(* IEC 61131-3 sources: CodesysTest/alpha/export/FBs/Components/BagOpenFingers/FB_BagOpenFingers.pou, 1 file *)

(* ---- FB_BagOpenFingers.pou.st ---- *)
(*#-#-#-#-#-#-#-#-#-#---Declaration---#-#-#-#-#-#-#-#-#-#-#-#-#*)

FUNCTION_BLOCK FB_BagOpenFingers EXTENDS FB_BaseComponent
VAR_INPUT
END_VAR
VAR_OUTPUT
    releaseOutput : BOOL;
	grabOutput : BOOL;
END_VAR
VAR
    _releaseCommand : BOOL;
    _grabCommand : BOOL;
END_VAR
(*#-#-#-#-#-#-#-#-#-#---Implementation---#-#-#-#-#-#-#-#-#-#-#-#-#*)

SUPER^();
releaseOutput := _releaseCommand AND enable;
grabOutput := _grabCommand AND enable;
